PROGRAM TEST2
VAR
	cbCommand : CommandBlockPos;
	
	fbRunCommand : RunCommandBlock;
	fbPower : MC_Power;
	
	state : WORD;
	
	transition : BOOL := FALSE;
	
	varWord:LWORD := 10000;
	varLREAL:LREAL := 0;
END_VAR

CASE state OF
	1:
	transition:=FALSE;
	fbRunCommand(ptBlock:= ADR(cbCommand), bDone=> transition);
	IF transition THEN
		state:=2;
	END_IF
	2:
	;
END_CASE

END_PROGRAM

(* stored: Version 1.1.0.1, ProductVersion 3.1.4022.10
   POU TEST2: Id {f8b57de7-b0e5-49ae-a899-350ad1b9c6c9}, SpecialFunc None *)
